Staubli VAL3: RefreshList.pgx

program RefreshList()
  local num l_ni
begin
  //

  if bListRefresh
    resize(sList,1,32)
    for l_ni=0 to 15
      sList[l_ni]="dIn"+toString("",l_ni+1)
      sList[l_ni+15]="dOut"+toString("",l_ni+1)
    endFor
  endIf

end
